// TIA Portal V18 export
FUNCTION "LGF_CalcCRC16" : Word   // FC10019, SCL
{ S7_Optimized_Access := 'TRUE' }
AUTHOR : Siemens_Industry_Support
FAMILY : LGF
NAME : LGF_CRC16
VERSION : 0.0.0.0
// stored: IsIECCheckEnabled true, SetENOAutomatically false
   VAR_INPUT
      initValue : Word;   // Start value with which the calculation is executed. If there is no need for start value - assign 16#00 / Startwert, mit dem die Berechnung durchgeführt wird. Wenn keinen Startwert notwendig ist - 16#00 zuweisen.
      mask : Word;   // Generator polynomial with which the calculation is executed. (Mask / CRC polynomial) / Generatorpolynom, mit dem die Berechnung durchgeführt wird. (Maske / CRC Polynom)
      noOfElements : UInt;   // Number of elements to be used in CRC calculation 0 = all elements / the whole array / Anzahl der Elemente, die in der CRC-Berechnung verwendet werden 0 = alle Elemente / das gesamte Array
   END_VAR
   VAR_IN_OUT
      "array" : Array[*] of Byte;   // Data stream for which the CRC value will be calculated. / Datenstrom, für den der CRC-Wert berechnet werden soll.
   END_VAR
   VAR_TEMP
      tempCRC : Word;   // Temp CRC checksum / Temp CRC Prüfsumme
      tempLowerLimit : DInt;   // Temp Lower limit of input array / Temp Untergrenze Eingangs Array
      tempUpperLimit : DInt;   // Temp Upper limit of input array / Temp Obergrenze Eingangs Array
      tempIndexArray : DInt;   // Temp Array schleifen Index / Temp array loop index
      tempIndexCRC : DInt;   // Temp CRC Schleifen Index / Temp CRC loop index
   END_VAR
   VAR CONSTANT
      SHIFT_ONE_BIT : UInt := 1;   // Shift the CRC Calculation by 1 bit / Schieben der CRC Berechnung um ein Bit
      SHIFT_ONE_BYTE : UInt := 8;   // Shift by 1 byte (= 8 bits) / Schieben um ein Byte (= 8 Bit)
      ARRAY_FIRST_DIMENSION : UInt := 1;   // First dimension in the Array / Erste Dimension im Array
      CRC_LOOP_LOWER_LIMIT : DInt := 0;   // Lower limit of CRC loop / Untere Grenze für die CRC Berechnungsschleife
      CRC_LOOP_UPPER_LIMIT : DInt := 7;   // Upper limit of CRC loop / Obere Grenze für die CRC Berechnungsschleife
      ERR_NO_OF_ELEMENTS : Word := 16#8400;   // Error: `noOfElements` exceeds the maximum number of array elements / Fehler aufgrund eines undefinierten Zustands in der Zustandsmaschine
      STATUS_NO_ERROR : Word := 16#0000;   // No error occurred in function call / Kein Fehler beim Aufruf der Funktion aufgetreten
   END_VAR
   // Ret_Val : Berechneter CRC-Wert (Rückgabewert der Funktion). / Calculated CRC value (return value of the function).
BEGIN
   REGION Block info header
     //===============================================================================
     // SIEMENS AG / (c)Copyright 2019
     //-------------------------------------------------------------------------------
     // Title:            LGF_CRC16
     // Comment/Function: This function makes a CRC calculation according
     //                   to the CRC-16 algorithm
     // Library/Family:   LGF (Library General Functions)
     // Author:           Siemens Digital Industry Support
     // Tested with:      CPU 1515F-2 PN FW:V2.6
     // Engineering:      TIA Portal V15.1 Update 2
     // Restrictions:     ENO disabled - no error handling, no failure possible
     // Requirements:     PLC (S7-1200 / S7-1500)
     //-------------------------------------------------------------------------------
     // Change log table:
     // Version  | Date       | Expert in charge       | Changes applied
     //----------|------------|------------------------|------------------------------
     // 01.00.00 03.07.2018  Siemens Industry Online Support
     //                      First released version
     // 01.00.01 17.08.2018  Siemens Industry Online Support
     //                      Upgrade: TIA V15 Update 2
     // 01.00.02 23.11.2018  Siemens Industry Online Support
     //                      Upgrade: TIA V15.1
     // 01.00.03 09.10.2019  Simatic Systems Support
     //                      Code refactoring, comments added
     // 03.00.00 23.04.2020  Simatic Systems Support
     //                      Set version to V3.0.0, harmonize the version of the whole library
     // 03.00.01 12.11.2020  Simatic Systems Support
     //                      Insert documentation
     //                      Assign default start values to optional inputs - `initValue`, `mask`
     // 03.01.00 14.04.2023  Simatic Systems Support
     //                      Add input `noOfElements` to assign length to be converted different from array size 
     //                      Add outputs `error` and `status` display a wrong assignment to `noOfElements`
     //=============================================================================
   END_REGION Block info header

   REGION DESCRIPTION
     (/**/)
   END_REGION DESCRIPTION

   REGION Initialization and input data processing
     // Defining initial value for algorithm
     #tempCRC := #initValue;
     // Input array size calculation
     #tempLowerLimit := LOWER_BOUND(ARR := #array, DIM := #ARRAY_FIRST_DIMENSION);
     #tempUpperLimit := UPPER_BOUND(ARR := #array, DIM := #ARRAY_FIRST_DIMENSION);

     // check paramter `noOfELements`, if gretaer than zero check if fits to array size
     IF #noOfElements > 0 THEN
         IF #noOfElements > (#tempUpperLimit - #tempLowerLimit + 1) THEN
         ENO := FALSE;
         #LGF_CalcCRC16 := #tempCRC;
         RETURN;
       ELSE
         #tempUpperLimit := #tempLowerLimit + #noOfElements - 1;
       END_IF;
     END_IF;
   END_REGION

   REGION CRC calculation
     FOR #tempIndexArray := #tempLowerLimit TO #tempUpperLimit DO
       // Perform division using XOR function for appropriate word in array (with shift byte into MSB of 16bit CRC)
         #tempCRC := #tempCRC XOR BYTE_TO_WORD(#array[#tempIndexArray]);

       FOR #tempIndexCRC := #CRC_LOOP_LOWER_LIMIT TO #CRC_LOOP_UPPER_LIMIT DO
         // Check if MSB is set
         IF #tempCRC.%X0 THEN
           // Shift left and perform division by mask polynomial using XOR function
           #tempCRC := SHR(IN := #tempCRC, N := #SHIFT_ONE_BIT) XOR #mask;
         ELSE
           // Shift left without division
           #tempCRC := SHR(IN := #tempCRC, N := #SHIFT_ONE_BIT);
         END_IF;
       END_FOR;

     END_FOR;
   END_REGION

   REGION Outputs assignment
       #LGF_CalcCRC16 := #tempCRC;
     ENO := TRUE;
   END_REGION
END_FUNCTION
